Yaskawa INFORM job: SIDE-A-UNCLAMP.JBI

/JOB
//NAME SIDE-A-UNCLAMP
///FOLDERNAME CLAMPUNCLAMP
//POS
///NPOS 0,0,0,0,0,0
//INST
///DATE 2021/09/30 12:19
///ATTR SC,RW
NOP
'**OPEN CLAMP SIDE-A**
'*********************
'OPEN CLAMP
DOUT OT#(138) OFF
DOUT OT#(137) ON
'OPEN POKEYOKE
DOUT OT#(140) OFF
DOUT OT#(139) ON
END
